TYPE E_PumpState :
(
pumpSTOPPED	:= 0,
pumpSTARTING	:= 1,
pumpRUNNING	:= 2,
pumpFAULT := 3,
pumpSTOPPING :=4
);
END_TYPE

(* stored: Version 1.1.0.1
   DUT E_PumpState: Id {cd10f6fd-e32a-457c-9058-4461bcc9d005} *)
